{attribute 'GeneratedUsingTerminal: EK1122-0000-0018'}
{attribute addProperty BoxType "EK1122-0000-0018"}
{attribute addProperty Id "Beckhoff_CUxxxxsub_EK1100EK1100_AB5A94672A_0001_CU1123_0000_0016A_0001_CU1123_0000_0016_E3575DAD124"}
{attribute addProperty CRC "4256383231"}
{attribute addProperty Size "126"}
TYPE Beckhoff_CUxxxxEK1122_FDB340FF EXTENDS EK1122_AB5A9467 :
STRUCT
	{attribute addProperty Name "Beckhoff_CUxxxxsub_EK1100"}
	{attribute addProperty PreviousPort "Beckhoff CUxxxxEK1122 : D"}
	Beckhoff_CUxxxxsub_EK1100 : EK1100_AB5A9467;
	{attribute addProperty Name "A_0001_CU1123_0000_0016"}
	{attribute addProperty PreviousPort "Beckhoff CUxxxxsub EK1100 : C"}
	A_0001_CU1123_0000_0016 : A_0001_CU1123_0000_0016_E3575DAD;
END_STRUCT
END_TYPE

(* stored: Version 1.2.0.0, ProductVersion 3.1.4024.9
   DUT Beckhoff_CUxxxxEK1122_FDB340FF: Id {c12208e2-ac7a-4792-a307-4ff7684693c4} *)
